(* IEC 61131-3 sources: CODESYS-IO-Visualization/CODESYS-IO-Visualization.fbsproj/Pi.device.xml.v3^/Plc Logic.plclogic.xml.v3^/Application.application.xml.v3^/Programs/Z_System, 3 files *)

(* ---- OnlineChangeDone.fn.st ---- *)
// Do not change the interface of this function!
// This function is implicitly generated by the 'Task Configuration' and handles an event triggered by the runtime system.
// See tab 'System Events' of the 'Task Configuration' editor.
FUNCTION OnlineChangeDone : DWORD
VAR_IN_OUT
	EventPrm: CmpApp.EVTPARAM_CmpApp;
END_VAR
VAR
END_VAR

Main_IO.Init := TRUE;

(* ---- PrepareStop.fn.st ---- *)
// Do not change the interface of this function!
// This function is implicitly generated by the 'Task Configuration' and handles an event triggered by the runtime system.
// See tab 'System Events' of the 'Task Configuration' editor.
FUNCTION PrepareStop : DWORD
VAR_IN_OUT
	EventPrm: CmpApp.EVTPARAM_CmpAppStop;
END_VAR
VAR
END_VAR

(* ---- StartDone.fn.st ---- *)
// Do not change the interface of this function!
// This function is implicitly generated by the 'Task Configuration' and handles an event triggered by the runtime system.
// See tab 'System Events' of the 'Task Configuration' editor.
FUNCTION StartDone : DWORD
VAR_IN_OUT
	EventPrm: CmpApp.EVTPARAM_CmpApp;
END_VAR
VAR
END_VAR

Main_IO.Init := TRUE;
